(* IEC 61131-3 sources: RL_MAR/experiments/comparison/llm4plc/results/gpt-4o-mini_20260506_100619/20260506_102811, 3 files *)

(* ---- generated_code_iteration_0.st ---- *)
ructured-text
START_ST
FUNCTION_BLOCK FB_CourseDifferenceControl
VAR_INPUT
    KOMPASS_GRAD : INT; // Input compass angle
    KURS : INT; // Input course angle
END_VAR
VAR_OUTPUT
    KURS_DIFF : INT; // Output difference between course and compass
END_VAR

// Logic to compute the difference
IF KOMPASS_GRAD < 0 THEN
    KURS_DIFF := 0;
ELSE
    KURS_DIFF := KURS - KOMPASS_GRAD;

    // Adjust KURS_DIFF if it exceeds the defined boundaries
    IF KURS_DIFF > 1800 THEN
        KURS_DIFF := KURS_DIFF - 3600;
    ELSIF KURS_DIFF < -1800 THEN
        KURS_DIFF := KURS_DIFF + 3600;
    END_IF;
END_IF;

END_FUNCTION_BLOCK

PROGRAM MAIN
VAR
    fbCourseDiffControl : FB_CourseDifferenceControl; // Instance of the function block
    KOMPASS_GRAD : INT; // Compass angle input
    KURS : INT; // Course angle input
END_VAR

// Call the function block with the inputs
fbCourseDiffControl(KOMPASS_GRAD := KOMPASS_GRAD, KURS := KURS);

// Use the output
KURS_DIFF := fbCourseDiffControl.KURS_DIFF;

END_PROGRAM
END_ST

(* ---- generated_code_iteration_1.st ---- *)
START_REASON
The errors in the original Structured Text (ST) code occurred due to the incorrect use of the PROGRAM structure. The feedback indicates that the `MAIN` section was defined as a PROGRAM, which cannot be instantiated like a function block. Additionally, the variable section used "END_VAR" correctly, but the overall structure needs to maintain the function block format without switching to a program. Therefore, I will convert the `MAIN` section into a function block and ensure that the code adheres to the required structure.
END_REASON

START_ST
FUNCTION_BLOCK FB_CourseDifferenceControl
VAR_INPUT
    KOMPASS_GRAD : INT; // Input compass angle
    KURS : INT; // Input course angle
END_VAR
VAR_OUTPUT
    KURS_DIFF : INT; // Output difference between course and compass
END_VAR

// Logic to compute the difference
IF KOMPASS_GRAD < 0 THEN
    KURS_DIFF := 0;
ELSE
    KURS_DIFF := KURS - KOMPASS_GRAD;

    // Adjust KURS_DIFF if it exceeds the defined boundaries
    IF KURS_DIFF > 1800 THEN
        KURS_DIFF := KURS_DIFF - 3600;
    ELSIF KURS_DIFF < -1800 THEN
        KURS_DIFF := KURS_DIFF + 3600;
    END_IF;
END_IF;

END_FUNCTION_BLOCK

FUNCTION_BLOCK FB_Main
VAR
    fbCourseDiffControl : FB_CourseDifferenceControl; // Instance of the function block
    KOMPASS_GRAD : INT; // Compass angle input
    KURS : INT; // Course angle input
END_VAR

// Call the function block with the inputs
fbCourseDiffControl(KOMPASS_GRAD := KOMPASS_GRAD, KURS := KURS);

// Use the output
KURS_DIFF := fbCourseDiffControl.KURS_DIFF;

END_FUNCTION_BLOCK
END_ST

(* ---- generated_code_iteration_2.st ---- *)
START_REASON
The errors in the original Structured Text (ST) code occurred because the variable `KURS_DIFF` was defined as an output in the `FB_CourseDifferenceControl` function block but was not properly accessed in the `FB_Main` function block. The output variable should be accessed through the instance of the function block. Additionally, the structure of the code needs to ensure that all variables are correctly defined and utilized within the function block context. I will ensure that the output variable is accessed correctly and that the overall structure adheres to the requirements.
END_REASON

START_ST
FUNCTION_BLOCK FB_CourseDifferenceControl
VAR_INPUT
    KOMPASS_GRAD : INT; // Input compass angle
    KURS : INT; // Input course angle
END_VAR
VAR_OUTPUT
    KURS_DIFF : INT; // Output difference between course and compass
END_VAR

// Logic to compute the difference
IF KOMPASS_GRAD < 0 THEN
    KURS_DIFF := 0;
ELSE
    KURS_DIFF := KURS - KOMPASS_GRAD;

    // Adjust KURS_DIFF if it exceeds the defined boundaries
    IF KURS_DIFF > 1800 THEN
        KURS_DIFF := KURS_DIFF - 3600;
    ELSIF KURS_DIFF < -1800 THEN
        KURS_DIFF := KURS_DIFF + 3600;
    END_IF;
END_IF;

END_FUNCTION_BLOCK

FUNCTION_BLOCK FB_Main
VAR
    fbCourseDiffControl : FB_CourseDifferenceControl; // Instance of the function block
    KOMPASS_GRAD : INT; // Compass angle input
    KURS : INT; // Course angle input
    KURS_DIFF : INT; // Local variable to store the output difference
END_VAR

// Call the function block with the inputs
fbCourseDiffControl(KOMPASS_GRAD := KOMPASS_GRAD, KURS := KURS);

// Use the output
KURS_DIFF := fbCourseDiffControl.KURS_DIFF;

END_FUNCTION_BLOCK
END_ST
